(* PLC project Unnamed, Unknown Unnamed 1 *)
(* stored: creationDateTime 2022-11-22T23:07:47, modificationDateTime 2022-11-22T23:17:10 *)

PROGRAM SafetyProgram
  VAR_INPUT
    StartButton : BOOL;
    StopButton : BOOL;
    DoorSensor : BOOL;
    ControlEnable : BOOL;
    ControlReference : BOOL;
  END_VAR
  VAR_OUTPUT
    MainBreaker : DINT;
    SecondaryBreaker : BOOL;
    DischargeBreaker : BOOL;
    RunLight : BOOL;
    EnabledLight : BOOL;
    StopLight : BOOL;
    ControllerStart : BOOL;
    ControllerRef : BOOL;
  END_VAR

END_PROGRAM

CONFIGURATION Config0
  RESOURCE Res0 ON PLC
    TASK task0(INTERVAL := T#20ms, PRIORITY := 0);
    PROGRAM instance0 WITH task0 : SafetyProgram;
  END_RESOURCE
END_CONFIGURATION
